FUNCTION F_Temp_Write_Set_Point : ST_Modbus_Send_Frame
VAR_INPUT
	Module_Number	:WORD;
	Write_Value		:WORD;
END_VAR
VAR
END_VAR

F_Temp_Write_Set_Point := F_Temp_Write_Value(Module_Number:=Module_Number,
											Command_Index:=2,
											Write_Value:=Write_Value);

END_FUNCTION

(* stored: Version 1.1.0.1
   POU F_Temp_Write_Set_Point: Id {13e9245b-ce18-4824-91fc-976f21622026}, SpecialFunc None *)
